# EPICS substitutions: iocApp/Db/galil_csmotors.substitutions
# $File: //ASP/Dev/SBS/4_Controls/4_3_Network_Infrastructure/4_3_1_Comms_Common_Services/sw/device_drivers/Galil/1-5/galilTestApp/Db/galil_motor_withwrappers.substitutions $
# $Revision: #3 $
# $DateTime: 2012/03/22 09:46:31 $
# $Author: cliftm $
#
# Description
# Substitution file for galil_motors.template
#
# This library is free software; you can redistribute it and/or
# modify it under the terms of the GNU Lesser General Public
# Licence as published by the Free Software Foundation; either
# version 2.1 of the Licence, or (at your option) any later version.
#
# This library is distributed in the hope that it will be useful,
# but WITHOUT ANY WARRANTY; without even the implied warranty of
# MERCHANTABILITY or FITNESS FOR A PARTICULAR PURPOSE.  See the GNU
# Lesser General Public Licence for more details.
#
# You should have received a copy of the GNU Lesser General Public
# Licence along with this library; if not, write to the Free Software
# Foundation, Inc., 51 Franklin St, Fifth Floor, Boston, MA 02110-1301 USA.
#
# Contact details:
# mark.clift@synchrotron.org.au
# 800 Blackburn Road, Clayton, Victoria 3168, Australia.
#

file "$(GALIL)/db/galil_motor-v6-10up.template"
{
pattern
# Coordinate system (CS) motors
# If real motors in CSAxis require backlash correction then NTM must be NO
# If only CSAxis requires backlash correction NTM can be any value
{ P,        M,          PORT,   ADDR, EGU, DESC, VELO,  VMAX, ACCL, BDST, BVEL,  BACC, MRES,  SREV, ERES,  PREC, DHLM,    DLLM,    OFF,   UEIP, RTRY, NTM,  PCOF, ICOF, DCOF}
{"$(DMC)", "$(VM1=I)", "Galil", 8,    mm,  "",   20,    20,    1,     0,     0,     5, .001,  1000, 0.001, 5,    42273.3, -42273.3, 0,       0,    0   , "NO",  0,    0,    0}
{"$(DMC)", "$(VM2=J)", "Galil", 9,    mm,  "",   20,    20,    1,     0,     0,     5, .001,  1000, 0.001, 5,    42273.3, -42273.3, 0,       0,    0   , "NO",  0,    0,    0}
{"$(DMC)", "$(VM3=K)", "Galil", 10,   mm,  "",   20,    20,    1,     0,     0,     5, .001,  1000, 0.001, 5,    42273.3, -42273.3, 0,       0,    0   , "NO",  0,    0,    0}
{"$(DMC)", "$(VM4=L)", "Galil", 11,   mm,  "",   20,    20,    1,     0,     0,     5, .001,  1000, 0.001, 5,    42273.3, -42273.3, 0,       0,    0   , "NO",  0,    0,    0}
{"$(DMC)", "$(VM5=M)", "Galil", 12,   mm,  "",   20,    20,    1,     0,     0,     5, .001,  1000, 0.001, 5,    42273.3, -42273.3, 0,       0,    0   , "NO",  0,    0,    0}
{"$(DMC)", "$(VM6=N)", "Galil", 13,   mm,  "",   20,    20,    1,     0,     0,     5, .001,  1000, 0.001, 5,    42273.3, -42273.3, 0,       0,    0   , "NO",  0,    0,    0}
{"$(DMC)", "$(VM7=O)", "Galil", 14,   mm,  "",   20,    20,    1,     0,     0,     5, .001,  1000, 0.001, 5,    42273.3, -42273.3, 0,       0,    0   , "NO",  0,    0,    0}
{"$(DMC)", "$(VM8=P)", "Galil", 15,   mm,  "",   20,    20,    1,     0,     0,     5, .001,  1000, 0.001, 5,    42273.3, -42273.3, 0,       0,    0   , "NO",  0,    0,    0}
}

# end
